(* IEC 61131-3 sources: uwecyber.github.io/cpss/resources/files, 3 files *)

(* ---- Bakery.st ---- *)
PROGRAM program0
  VAR
    I_Start AT %IX100.1 : BOOL;
    I_Stop AT %IX100.2 : BOOL;
  END_VAR
  VAR
    V_MixingProcess : BOOL;
    V_SplittingProcess : BOOL;
    V_Stop : BOOL;
  END_VAR
  VAR
    Conveyer_Flour AT %QX100.0 : BOOL;
    Conveyer_Yeast AT %QX100.1 : BOOL;
    Conveyer_SS AT %QX100.2 : BOOL;
    Conveyer_Additives AT %QX100.3 : BOOL;
    Conveyer_Oil AT %QX100.4 : BOOL;
    Conveyer_Water AT %QX100.5 : BOOL;
    SpawnA_1 AT %QX100.6 : BOOL;
    SpawnA_2 AT %QW100.1 : INT;
    SpawnA_3 AT %QW101.1 : INT;
    SpawnB_1 AT %QX102.4 : BOOL;
    SpawnB_2 AT %QW102.1 : INT;
    SpawnB_3 AT %QW103.1 : INT;
    FlourDiff AT %IX100.3 : BOOL;
    YeastDiff AT %IX100.4 : BOOL;
    MixingDiff AT %IX100.5 : BOOL;
    SSDiff AT %IX100.6 : BOOL;
    AdditivesDiff AT %IX100.7 : BOOL;
    DrymixingDiff AT %IX101.0 : BOOL;
    OilDiff AT %IX101.1 : BOOL;
    WaterDiff AT %IX101.2 : BOOL;
    WetmixingDiff AT %IX101.3 : BOOL;
    SplittingDiff AT %IX101.4 : BOOL;
    ProofingOvenDiff AT %IX101.5 : BOOL;
    BakingOvenDiff AT %IX101.6 : BOOL;
    EmergencyStop AT %IX101.7 : BOOL;
    FlourStop AT %QX100.7 : BOOL;
    YeastStop AT %QX101.0 : BOOL;
    MixingConveyor AT %QX101.1 : BOOL;
    SSStop AT %QX101.2 : BOOL;
    AdditivesStop AT %QX101.3 : BOOL;
    DrymixingConveyor AT %QX101.4 : BOOL;
    DrymixingStop AT %QX101.5 : BOOL;
    OilStop AT %QX101.6 : BOOL;
    WaterStop AT %QX101.7 : BOOL;
    WetMixingConveyor AT %QX102.0 : BOOL;
    WetMixingStop AT %QX102.1 : BOOL;
    SplittingConveyor AT %QX102.2 : BOOL;
    Split AT %QX102.3 : BOOL;
    ProofingOvenConveyor AT %QX102.5 : BOOL;
    ConnectorConveyor AT %QX102.6 : BOOL;
    BakingOvenConveyor AT %QX102.7 : BOOL;
    StopConveyor AT %QX103.0 : BOOL;
    Endmixing AT %QX103.1 : BOOL;
  END_VAR
  VAR
    RS1 : RS;
    RS2 : RS;
    RS3 : RS;
    RS4 : RS;
    RS5 : RS;
    RS6 : RS;
    RS7 : RS;
    RS8 : RS;
    RS9 : RS;
    TP0 : TP;
    TP1 : TP;
    TP2 : TP;
    TP3 : TP;
    TP4 : TP;
    TP5 : TP;
    TP6 : TP;
    TP7 : TP;
    TP8 : TP;
    TP9 : TP;
    TP10 : TP;
    TON0 : TON;
    RS10 : RS;
    RS11 : RS;
    RS12 : RS;
    TP11 : TP;
    TP12 : TP;
    TON1 : TON;
    RS0 : RS;
    RS13 : RS;
    TON2 : TON;
    NOT137_OUT : BOOL;
    NOT133_OUT : BOOL;
    NOT48_OUT : BOOL;
    NOT54_OUT : BOOL;
    NOT52_OUT : BOOL;
    NOT55_OUT : BOOL;
    NOT135_OUT : BOOL;
  END_VAR

  SpawnA_1 := V_MixingProcess;
  SpawnA_2 := 0000000000000000;
  SpawnB_1 := V_SplittingProcess;
  SpawnA_3 := 0000000000000001;
  SpawnB_3 := 0000000000000000;
  NOT137_OUT := NOT(I_Stop);
  RS1(S := I_Start, R1 := NOT137_OUT);
  V_MixingProcess := RS1.Q1;
  SpawnB_2 := 0000000000000001;
  RS2(S := I_Start, R1 := NOT137_OUT);
  Conveyer_Flour := RS2.Q1;
  NOT133_OUT := NOT(I_Stop);
  V_Stop := NOT133_OUT;
  RS3(S := I_Start, R1 := NOT137_OUT);
  Conveyer_Yeast := RS3.Q1;
  NOT48_OUT := NOT(EmergencyStop);
  V_Stop := NOT48_OUT;
  NOT54_OUT := NOT(I_Stop);
  RS11(S := I_Start, R1 := NOT54_OUT);
  ConnectorConveyor := RS11.Q1;
  NOT52_OUT := NOT(I_Stop);
  RS5(S := I_Start, R1 := NOT52_OUT);
  Conveyer_SS := RS5.Q1;
  RS10(S := I_Start, R1 := NOT54_OUT);
  StopConveyor := RS10.Q1;
  RS4(S := I_Start, R1 := NOT52_OUT);
  Conveyer_Additives := RS4.Q1;
  RS12(S := I_Start, R1 := NOT54_OUT);
  Endmixing := RS12.Q1;
  RS6(S := I_Start, R1 := NOT52_OUT);
  Conveyer_Oil := RS6.Q1;
  NOT55_OUT := NOT(I_Stop);
  RS8(S := I_Start, R1 := NOT55_OUT);
  Conveyer_Water := RS8.Q1;
  RS7(S := I_Start, R1 := NOT55_OUT);
  DrymixingConveyor := RS7.Q1;
  RS9(S := I_Start, R1 := NOT55_OUT);
  WetMixingConveyor := RS9.Q1;
  TP0(IN := FlourDiff, PT := T#12S);
  FlourStop := TP0.Q;
  TP1(IN := YeastDiff, PT := T#6S);
  YeastStop := TP1.Q;
  TP2(IN := MixingDiff, PT := T#15S);
  MixingConveyor := TP2.Q;
  TP3(IN := SSDiff, PT := T#8S);
  SSStop := TP3.Q;
  TP4(IN := AdditivesDiff, PT := T#6S);
  AdditivesStop := TP4.Q;
  TP5(IN := DrymixingDiff, PT := T#14S);
  DrymixingStop := TP5.Q;
  TP6(IN := OilDiff, PT := T#7S);
  OilStop := TP6.Q;
  TP7(IN := WaterDiff, PT := T#9S);
  WaterStop := TP7.Q;
  TP8(IN := WetmixingDiff, PT := T#45S);
  WetMixingStop := TP8.Q;
  TP9(IN := WetmixingDiff, PT := T#65S);
  SplittingConveyor := TP9.Q;
  TP10(IN := SplittingDiff, PT := T#5S);
  Split := TP10.Q;
  TON0(IN := TP10.Q, PT := T#2S);
  V_SplittingProcess := TON0.Q;
  NOT135_OUT := NOT(ProofingOvenDiff);
  TP11(IN := NOT135_OUT, PT := T#25S);
  ProofingOvenConveyor := TP11.Q;
  TP12(IN := BakingOvenDiff, PT := T#25S);
  BakingOvenConveyor := TP12.Q;
  RS0(S := BakingOvenDiff, R1 := V_Stop);
  TON1(IN := RS0.Q1, PT := T#30S);
  TON2(IN := TON1.Q, PT := T#5S);
  RS13(S := TON1.Q, R1 := TON2.Q);
  V_Stop := RS13.Q1;
END_PROGRAM

CONFIGURATION Config0

  RESOURCE Res0 ON PLC
    TASK task0(INTERVAL := T#20ms,PRIORITY := 0);
    PROGRAM instance0 WITH task0 : program0;
  END_RESOURCE
END_CONFIGURATION

(* ---- CircularScene.st ---- *)
PROGRAM conveyors
  VAR
    Start_Button AT %IX100.0 : BOOL;
    Stop_Button AT %IX100.1 : BOOL;
    TT1_Limit90Left AT %IX100.3 : BOOL;
    TT1_FrontLim AT %IX100.4 : BOOL;
    TT1_Limit0 AT %IX100.5 : BOOL;
    TT2_Limit90Lef AT %IX100.6 : BOOL;
    TT2_FrontLim AT %IX100.7 : BOOL;
    TT2_Limit0 AT %IX101.0 : BOOL;
    Run AT %QX107.0 : BOOL;
    Conveyor1 AT %QX100.0 : BOOL;
    Conveyor2 AT %QX100.1 : BOOL;
    Conveyor3 AT %QX100.2 : BOOL;
    Conveyor4 AT %QX100.3 : BOOL;
    Conveyor5 AT %QX100.4 : BOOL;
    Conveyor6 AT %QX100.5 : BOOL;
    CurvedConveryor1 AT %QX100.6 : BOOL;
    CurvedConveyor2 AT %QX100.7 : BOOL;
    TT1_Turn AT %QX101.0 : BOOL;
    TT1_RollForward AT %QX101.1 : BOOL;
    RS1 AT %QX101.2 : BOOL;
    TT2_Turn AT %QX101.3 : BOOL;
    TT2_RollForward AT %QX101.4 : BOOL;
    RS2 AT %QX101.5 : BOOL;
  END_VAR

  Run := Stop_Button AND (Run OR Start_Button);
  Conveyor1 := Run;
  Conveyor2 := Run;
  Conveyor3 := Run;
  Conveyor4 := Run;
  Conveyor5 := Run;
  Conveyor6 := Run;
  CurvedConveryor1 := Run;
  CurvedConveyor2 := Run;
  TT1_RollForward := NOT(TT1_FrontLim AND Run);
  RS1 := TT1_FrontLim AND Run;
  TT1_Turn := TT1_Limit0 AND RS1 AND Run;
  TT1_Turn := NOT(NOT(TT1_FrontLim) AND Run);
  RS1 := NOT(TT1_Limit0 AND NOT(TT1_FrontLim) AND Run);
  TT1_RollForward := TT1_Limit0 AND NOT(TT1_FrontLim) AND Run OR TT1_Limit90Left AND Run;
  TT2_RollForward := NOT(TT2_FrontLim AND Run);
  RS2 := TT2_FrontLim AND Run;
  TT2_Turn := TT2_Limit0 AND RS2 AND Run;
  TT2_Turn := NOT(NOT(TT2_FrontLim) AND Run);
  RS2 := NOT(TT2_Limit0 AND NOT(TT2_FrontLim) AND Run);
  TT2_RollForward := TT2_Limit0 AND NOT(TT2_FrontLim) AND Run OR TT2_Limit90Lef AND Run;
END_PROGRAM

CONFIGURATION Config0

  RESOURCE Res0 ON PLC
    TASK task0(INTERVAL := T#20ms,PRIORITY := 0);
    PROGRAM instance0 WITH task0 : conveyors;
  END_RESOURCE
END_CONFIGURATION

(* ---- WaterTreatment.st ---- *)
PROGRAM Main
  VAR
    I_PbFill AT %IX100.1 : BOOL;
    O_FillValve AT %QX100.0 : BOOL;
    O_DischargeValve AT %QX100.1 : BOOL;
  END_VAR
  VAR
    Filling : BOOL;
    Discharging : BOOL;
    FillDone : BOOL;
    Purify_Done1 : BOOL;
    Purify_Done2 : BOOL;
    Purify_Done3 : BOOL;
    Purify_Done4 : BOOL;
    Restart : BOOL;
  END_VAR
  VAR
    PH_Level AT %QW101.1 : INT;
    Chlorine_Level AT %QW100.1 : INT;
  END_VAR
  VAR
    TON0 : TON;
    RS0 : RS;
    TON1 : TON;
    RS1 : RS;
    R_TRIG0 : R_TRIG;
    RS2 : RS;
    TON2 : TON;
    CTU0 : CTU;
    TON3 : TON;
    CTU1 : CTU;
    TON4 : TON;
    CTU2 : CTU;
    TON5 : TON;
    CTU3 : CTU;
    TON6 : TON;
    TON7 : TON;
    TON8 : TON;
    TON9 : TON;
    OR50_OUT : BOOL;
    NOT3_OUT : BOOL;
    AND5_OUT : BOOL;
    R_TRIG1 : R_TRIG;
    R_TRIG2 : R_TRIG;
    ADD60_OUT : INT;
    R_TRIG3 : R_TRIG;
    R_TRIG4 : R_TRIG;
    ADD61_OUT : INT;
    ADD62_OUT : INT;
    SUB67_OUT : INT;
    NOT17_OUT : BOOL;
    AND19_OUT : BOOL;
  END_VAR

  R_TRIG0(CLK := I_PbFill);
  OR50_OUT := OR(Restart, R_TRIG0.Q);
  NOT3_OUT := NOT(Discharging);
  AND5_OUT := AND(OR50_OUT, NOT3_OUT);
  TON0(IN := Filling, PT := T#70S);
  RS0(S := AND5_OUT, R1 := TON0.Q);
  Filling := RS0.Q1;
  FillDone := TON0.Q;
  RS2(S := FillDone, R1 := Purify_Done4);
  TON2(IN := RS2.Q1, PT := T#2S);
  R_TRIG1(CLK := TON2.Q);
  CTU0(CU := R_TRIG1.Q, R := Purify_Done1, PV := 1);
  TON3(IN := RS2.Q1, PT := T#4S);
  R_TRIG2(CLK := TON3.Q);
  CTU1(CU := R_TRIG2.Q, R := Purify_Done2, PV := 1);
  ADD60_OUT := ADD(CTU0.CV, CTU1.CV);
  TON4(IN := RS2.Q1, PT := T#6S);
  R_TRIG3(CLK := TON4.Q);
  CTU2(CU := R_TRIG3.Q, R := Purify_Done3, PV := 1);
  TON5(IN := RS2.Q1, PT := T#8S);
  R_TRIG4(CLK := TON5.Q);
  CTU3(CU := R_TRIG4.Q, R := Purify_Done4, PV := 1);
  ADD61_OUT := ADD(CTU2.CV, CTU3.CV);
  ADD62_OUT := ADD(ADD60_OUT, ADD61_OUT);
  Chlorine_Level := ADD62_OUT;
  SUB67_OUT := SUB(7, ADD61_OUT);
  PH_Level := SUB67_OUT;
  TON6(IN := CTU3.Q, PT := T#8S);
  Purify_Done1 := TON6.Q;
  TON7(IN := TON6.Q, PT := T#2S);
  Purify_Done2 := TON7.Q;
  TON8(IN := TON7.Q, PT := T#2S);
  Purify_Done3 := TON8.Q;
  NOT17_OUT := NOT(Filling);
  AND19_OUT := AND(Purify_Done4, NOT17_OUT);
  TON1(IN := Discharging, PT := T#90S);
  RS1(S := AND19_OUT, R1 := TON1.Q);
  Discharging := RS1.Q1;
  TON9(IN := TON8.Q, PT := T#2S);
  Purify_Done4 := TON9.Q;
  Restart := TON1.Q;
  O_FillValve := Filling;
  O_DischargeValve := Discharging;
END_PROGRAM

CONFIGURATION Config0

  RESOURCE Res0 ON PLC
    TASK task0(INTERVAL := T#20ms,PRIORITY := 0);
    PROGRAM instance0 WITH task0 : Main;
  END_RESOURCE
END_CONFIGURATION
